// TIA Portal V17 program export: 2 tag tables, 0 data types, 1 data blocks, 3 code blocks (in call order from the OBs), 1 instance data blocks

VAR_GLOBAL   // PLC tag table "Default tag table"
   System_Byte AT %MB1 : Byte;
   FirstScan AT %M1.0 : Bool;
   DiagStatusUpdate AT %M1.1 : Bool;
   AlwaysTRUE AT %M1.2 : Bool;
   AlwaysFALSE AT %M1.3 : Bool;
   Clock_Byte AT %MB0 : Byte;
   Clock_10Hz AT %M0.0 : Bool;
   Clock_5Hz AT %M0.1 : Bool;
   "Clock_2.5Hz" AT %M0.2 : Bool;
   Clock_2Hz AT %M0.3 : Bool;
   "Clock_1.25Hz" AT %M0.4 : Bool;
   Clock_1Hz AT %M0.5 : Bool;
   "Clock_0.625Hz" AT %M0.6 : Bool;
   "Clock_0.5Hz" AT %M0.7 : Bool;
END_VAR

VAR_GLOBAL   // PLC tag table "IO"
   IB_0 AT %IB0 : Byte;
   IB_1 AT %IB1 : Byte;
   QB_0 AT %QB0 : Byte;
   QB_1 AT %QB1 : Byte;
   AQW_80 AT %QW80 : Word;
   AIW_64 AT %IW64 : Word;
   AIW_65 AT %IW66 : Word;
END_VAR

DATA_BLOCK "Internal"   // DB1
{ S7_Optimized_Access := 'TRUE' }
VERSION : 0.1
// stored: AutoNumber true, DBAccessibleFromOPCUA true, IsOnlyStoredInLoadMemory false, IsRetainMemResEnabled false, IsWriteProtectedInAS false, MemoryReserve 100
   VAR
      Start : Bool;
      Stop : Bool;
   END_VAR
BEGIN
END_DATA_BLOCK

ORGANIZATION_BLOCK "Main"   // OB1, LAD, ProgramCycle
TITLE = "Main Program Sweep (Cycle)"
{ S7_Optimized_Access := 'TRUE' }
VERSION : 0.1
// stored: AutoNumber true, IsIECCheckEnabled false, SetENOAutomatically false
   VAR_INPUT
      Initial_Call : Bool;   // Initial call of this OB
      Remanence : Bool;   // =True, if remanent data are available
   END_VAR
   VAR_TEMP
      Analog_value : Real;
   END_VAR
BEGIN

REGION Network 1
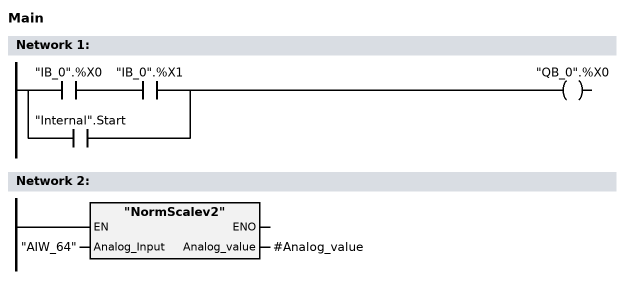
   RUNG wire#powerrail
      Contact( "IB_0".%X0 )
      Contact( "IB_0".%X1 )
      wire#w1
      Coil( "QB_0".%X0 )
   END_RUNG
   RUNG wire#powerrail
      Contact( "Internal".Start )
   END_RUNG wire#w1
   // the same network as SCL:
   "QB_0".%X0 := ("IB_0".%X0 AND "IB_0".%X1) OR "Internal".Start;
END_REGION

REGION Network 2
   RUNG wire#powerrail
      "NormScalev2"(Analog_Input := "AIW_64", Analog_value => #Analog_value)
   END_RUNG
   // the same network as SCL:
   "NormScalev2"(Analog_Input := "AIW_64", Analog_value => #Analog_value);
END_REGION
END_ORGANIZATION_BLOCK

FUNCTION "NormScalev2" : Void   // FC1, LAD
{ S7_Optimized_Access := 'TRUE' }
VERSION : 0.1
// stored: AutoNumber true, IsIECCheckEnabled false, SetENOAutomatically false, UDAEnableTagReadback false
   VAR_INPUT
      Analog_Input : UInt;
   END_VAR
   VAR_OUTPUT
      Analog_value : Real;
   END_VAR
   VAR_TEMP
      norm_analog_input : Real;
   END_VAR
   VAR CONSTANT
      Upper_int : UInt := 27648;
      Lower_int : UInt := 0;
      Upper_Real : Real := 100.0;
      Lower_Real : Real := 0.0;
   END_VAR
BEGIN

REGION Network 1
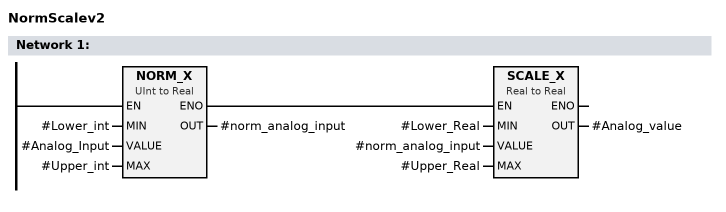
   RUNG wire#powerrail
      { S7_Templates := "[SrcType := UInt, DestType := Real]" } Normalize(min := #Lower_int, value := #Analog_Input, max := #Upper_int, out => #norm_analog_input)
      { S7_Templates := "[SrcType := Real, DestType := Real]" } Scale(min := #Lower_Real, value := #norm_analog_input, max := #Upper_Real, out => #Analog_value)
   END_RUNG
   // the same network as SCL:
   #norm_analog_input := NORM_X(MIN := #Lower_int, VALUE := #Analog_Input, MAX := #Upper_int);
   #Analog_value := SCALE_X(MIN := #Lower_Real, VALUE := #norm_analog_input, MAX := #Upper_Real);
END_REGION
END_FUNCTION

FUNCTION_BLOCK "FB_Testblok"
{ S7_Optimized_Access := 'TRUE' }
VERSION : 0.1
   VAR_INPUT 
      Input_Int : Int;
   END_VAR

   VAR_OUTPUT 
      Output_Real : Real;
   END_VAR

   VAR_TEMP 
      NormVal : Real;
   END_VAR


BEGIN
	#NormVal:=NORM_X_REAL(MIN := 0, VALUE := #Input_Int, MAX := 27648);
	#Output_Real:=SCALE_X_REAL(MIN := 0.0, VALUE := #NormVal, MAX := 100.0);
	
END_FUNCTION_BLOCK

DATA_BLOCK "FB_Testblok_DB"   // DB1
VERSION : 0.1
// stored: AutoNumber true, DBAccessibleFromOPCUA true, InstanceOfName FB_Testblok, InstanceOfType FB
"FB_Testblok"
BEGIN
END_DATA_BLOCK
